Staubli VAL3: encodeStatus.pgx

public program encodeStatus()
begin
  // Copyright (c) 2016, Ocado Technology - Robotics Research Team
  //
  // Licensed under the Apache License, Version 2.0 (the "License");
  // you may not use this file except in compliance with the License.
  // You may obtain a copy of the License at
  //
  //     http://www.apache.org/licenses/LICENSE-2.0
  //
  // Unless required by applicable law or agreed to in writing, software
  // distributed under the License is distributed on an "AS IS" BASIS,
  // WITHOUT WARRANTIES OR CONDITIONS OF ANY KIND, either express or implied.
  // See the License for the specific language governing permissions and
  // limitations under the License.



  // encode 'prefix' and 'header'
  call encPrefixHeader(rosStatusMsg.prefix, rosStatusMsg.header)

  // encode variables of body message (data)
  toBinary(rosStatusMsg.robotStatus.nDrivesPowered,1,"-4l",rosStatusMsg.body.nData)
  toBinary(rosStatusMsg.robotStatus.nEStopped,1,"-4l",rosStatusMsg.body.nData[4])
  toBinary(rosStatusMsg.robotStatus.nErrorCode,1,"-4l",rosStatusMsg.body.nData[8])
  toBinary(rosStatusMsg.robotStatus.nInError,1,"-4l",rosStatusMsg.body.nData[12])
  toBinary(rosStatusMsg.robotStatus.nInMotion,1,"-4l",rosStatusMsg.body.nData[16])
  toBinary(rosStatusMsg.robotStatus.nMode,1,"-4l",rosStatusMsg.body.nData[20])
  toBinary(rosStatusMsg.robotStatus.nMotionPossible,1,"-4l",rosStatusMsg.body.nData[24])
  toBinary(rosStatusMsg.robotStatus.nTrajComplete,1,"-4l",rosStatusMsg.body.nData[28])
end
